// TIA Portal V18 export
TYPE "MEStoPLC_PrintExchange"
// stored: IsFailsafeCompliant false
   STRUCT
      "M-PrintDataDone" : Bool;   // 打刻数据下发完成表示
      "M-PrintDataOK" : Bool;   // 打刻数据下发完成表示OK
      "M-PrintDataNG" : Bool;   // 打刻数据下发完成表示NG
      "M-PrintData" : Array[1..10] of String[48];   // 打刻数据，Print1-10总长500
      "M-PrintDataErrCode" : Int;   // 【预留】“M-ErrorMsg”失效的时候启用
      "M-PrintDataErrMsg" : String[98];   // 打印请求Mes标志位收到后，如果Mes对请求的数据校验有异常，写入相应中文字符串，M-PrintDataDone信号超时后将中文字符串显示到HMI
      Reserve : Array[1..396] of Byte;   // 打印打刻预留
   END_STRUCT;
END_TYPE
